FUNCTION_BLOCK FB_LightOnCommand IMPLEMENTS I_Command
VAR_INPUT
END_VAR
VAR_OUTPUT
END_VAR
VAR
	// Reference to the Light that should be switched on.
	iLight: I_Switchable;
END_VAR

METHOD Execute
IF (iLight <> 0) THEN
	THIS^.iLight.On();
END_IF
END_METHOD

METHOD FB_init : BOOL
VAR_INPUT
	bInitRetains : BOOL; // if TRUE, the retain variables are initialized (warm start / cold start)
	bInCopyCode : BOOL;  // if TRUE, the instance afterwards gets moved into the copy code (online change)
	iSwitchable : I_Switchable;
END_VAR
IF (iSwitchable <> 0) THEN
	THIS^.iLight := iSwitchable;
END_IF
END_METHOD

END_FUNCTION_BLOCK

(* stored: Version 1.1.0.1, ProductVersion 3.1.4024.5
   POU FB_LightOnCommand: Id {55ce3f02-0d03-4749-b749-2d01dc21a580}, SpecialFunc None
   Method Execute: Id {0a7472be-59a0-4e42-9999-69f8252c93a8}
   Method FB_init: Id {5d5c2768-1430-4b4c-b874-c6c297050f63} *)
